FUNCTION_BLOCK ASRT_MERGE_2 (* MERGE 2 ASRT into 1 ASRT (generic FB) *)
  (* Standard: 61499-2; Description: Copyright (c) 2026 Meisterschulen am Ostbahnhof This program and the accompanying materials are made available under the terms of the Eclipse Public License 2.0 which is available at https://www.eclipse.org/legal/epl-2.0/ SPDX-License-Identifier: EPL-2.0 *)
  (* Version 1.0, 2026-09-06, Franz Höpfinger, Meisterschulen am Ostbahnhof *)
  PACKAGE adapter::events::unidirectional;
  IMPORT eclipse4diac::core::GenericClassName;
  {SET_ATTRIBUTE(eclipse4diac::core::GenericClassName, 'GEN_ASRT_MERGE')}
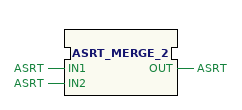
  SOCKETS
    IN1 : adapter::types::unidirectional::ASRT;
    IN2 : adapter::types::unidirectional::ASRT;
  END_SOCKETS
  PLUGS
    OUT : adapter::types::unidirectional::ASRT;
  END_PLUGS
END_FUNCTION_BLOCK
